SUBAPPLICATION mapping_Uebung_034a1_Q1 (* Numeric Value Input auf PWM Ausgang *)
  (* Standard: 61499-2; Description: Copyright (c) 2023 Meisterschulen am Ostbahnhof This program and the accompanying materials are made available under the terms of the Eclipse Public License 2.0 which is available at https://www.eclipse.org/legal/epl-2.0/ SPDX-License-Identifier: EPL-2.0 *)
  (* Version 1.0, 2023-10-23, Franz Höpfinger, Meisterschulen am Ostbahnhof *)
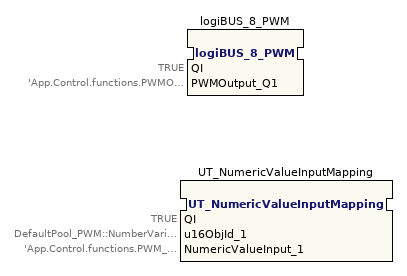
  FBS
    logiBUS_8_PWM : logiBUS_8_PWM(QI := TRUE, PWMOutput_Q1 := 'App.Control.functions.PWMOutput_Q1');
    UT_NumericValueInputMapping : UT_NumericValueInputMapping(QI := TRUE, u16ObjId_1 := DefaultPool_PWM::NumberVariable_PWM_Value, NumericValueInput_1 := 'App.Control.functions.PWM_Value');
  END_FBS
END_SUBAPPLICATION
